// TIA Portal V17 export
// export: Created 2021-12-03T08:12:53.7025583Z, ExportSetting WithDefaults, DisplayName Totally Integrated Automation Portal, DisplayVersion V17, DisplayName TIA Portal Openness, DisplayVersion V17, DisplayName TIA Portal Version Control Interface, DisplayVersion V17, DisplayName STEP 7 Professional, DisplayVersion V17, DisplayName STEP 7 Safety, DisplayVersion V17, DisplayName WinCC Advanced, DisplayVersion V17
DATA_BLOCK "GDB_HmiLog"   // DB1005
VERSION : 0.1
// stored: AutoNumber false, IsOnlyStoredInLoadMemory false, IsWriteProtectedInAS false
   VAR
      SafetyPer : Word;   // Условия для закрытия периметра
      ScanSeqCond : Word;   // Условия для запуска сканирования
      Alarm_CirBrk24VFb : Word;
      Alarm_CirBrk220VFb : Word;
      Alarm_CirBrk380VFb : Word;
      Alarm_EstpBtn_Mon : Word;
      Alarm_ContactorError : Word;
      ScanSeqFlt : Word;   // Ошибки последовательности сканирования
   END_VAR
BEGIN
END_DATA_BLOCK
